// TIA Portal project "VisionSensorKonveyorBandSistemi" (V17)
// Vorlageprojekt für das Buch mit Zielsystem S7-1200

(* hardware
DEVICE "S7-1200-Station_1"  S7-1200 Station
   slot 0: "Baugruppenträger_0"  Rack  V1.0
   slot 1: "PLC_1"  CPU 1211C DC/DC/DC  6ES7 211-1AE40-0XB0  V4.1
*)

// ===== PLC "PLC_1"  CPU 1211C DC/DC/DC =====

VAR_GLOBAL   // PLC tag table "Standard-Variablentabelle"
   "ENTRY CONVEYOR" AT %A0.0 : Bool;
   "EXİT" AT %E0.0 : Bool;
   "START PB" AT %E0.1 : Bool;
   "AUTO MANUAL" AT %I0.5 : Bool;
   "MANUAL" AT %M0.1 : Bool;
   "AUTO" AT %M0.0 : Bool;
   "ONS" AT %M1.1 : Bool;
   "START ONS" AT %M0.3 : Bool;
   "STOP PB" AT %I0.3 : Bool;
   "Tag_3" AT %I0.4 : Bool;
   "RUN MODE" AT %M0.4 : Bool;
   "START LIGHT" AT %Q1.1 : Bool;
   "STOP LIGHT" AT %Q1.3 : Bool;
   "RESET PB" AT %I0.2 : Bool;
   "RESET" AT %M0.2 : Bool;
   "RESET LIGHT" AT %Q1.2 : Bool;
   "VİSİON SENSOR" AT %IW104 : Int;
   "VİSİON SENSOR ARALIK" AT %M1.0 : Bool;
   "STOP ENTRY CONVEYOR" AT %M1.2 : Bool;
   "PRODUCT BLUE OR GREEN" AT %M0.5 : Bool;
   "BLUE BASE OR LID" AT %M0.6 : Bool;
   "GREEN BASE OR LİD" AT %M0.7 : Bool;
   "SORTER 2 BELT" AT %Q0.6 : Bool;
   "SORTER 2TURN" AT %Q0.5 : Bool;
   "Tag_2" AT %QW32 : Int;
   "EXİT CONVEYOR" AT %Q0.2 : Bool;
   "SORTER 1 BELT" AT %Q0.4 : Bool;
   "SORTER 1 TURN" AT %Q0.3 : Bool;
   "Tag_1" AT %QW30 : Int;
   "SORTER 3 BELT" AT %Q1.0 : Bool;
   "SORTER 3 TURN" AT %Q0.7 : Bool;
   "Tag_4" AT %QW34 : Int;
   "VISION SENSOR" AT %IW30 : Word;
END_VAR

// folder: System blocks/Program resources

DATA_BLOCK "IEC_Timer_0_DB"   // DB1
{ S7_Optimized_Access := 'TRUE' }
AUTHOR : Simatic
FAMILY : IEC
NAME : IEC_TMR
VERSION : 1.0
// stored: InstanceOfName IEC_TIMER
"IEC_TIMER"
BEGIN
END_DATA_BLOCK

DATA_BLOCK "IEC_Timer_0_DB_1"   // DB2
{ S7_Optimized_Access := 'TRUE' }
AUTHOR : Simatic
FAMILY : IEC
NAME : IEC_TMR
VERSION : 1.0
// stored: InstanceOfName IEC_TIMER
"IEC_TIMER"
BEGIN
END_DATA_BLOCK

DATA_BLOCK "IEC_Counter_0_DB"   // DB3
{ S7_Optimized_Access := 'TRUE' }
AUTHOR : Simatic
FAMILY : IEC
NAME : CNTR
VERSION : 1.0
// stored: InstanceOfName IEC_COUNTER
"IEC_COUNTER"
BEGIN
END_DATA_BLOCK

DATA_BLOCK "IEC_Counter_0_DB_1"   // DB4
{ S7_Optimized_Access := 'TRUE' }
AUTHOR : Simatic
FAMILY : IEC
NAME : CNTR
VERSION : 1.0
// stored: InstanceOfName IEC_COUNTER
"IEC_COUNTER"
BEGIN
END_DATA_BLOCK

DATA_BLOCK "IEC_Counter_0_DB_2"   // DB5
{ S7_Optimized_Access := 'TRUE' }
AUTHOR : Simatic
FAMILY : IEC
NAME : CNTR
VERSION : 1.0
// stored: InstanceOfName IEC_COUNTER
"IEC_COUNTER"
BEGIN
END_DATA_BLOCK

// folder: (top level)

FUNCTION "MHJ-PLC-Lab-Function-S71200" : Void   // FC9000, SCL
{ S7_Optimized_Access := 'TRUE' }
VERSION : 0.1
   VAR_TEMP
      rdTimeReturn : Int;
      outputTime : DTL;
      SyncVal : Byte;
      forVal : Int;
      forVal_2 : Int;
      Value : Byte;
   END_VAR
   VAR CONSTANT
      CompVal : Byte := 16#34;
      Value_01 : Byte := 16#11;
      Value_01_DW : DWord := 16#A165_D992;
      Value_02_DW : DWord := 16#58BE_4401;
   END_VAR
BEGIN

   #Value:=PEEK(area := 16#82,
        dbNumber := 0,
        byteOffset := 511);
   #Value := #Value + 1;

   POKE(area := 16#82,
        dbNumber := 0,
        byteOffset := 511,
        value := #Value);

   POKE(area:=16#81,
        dbNumber:=0,
        byteOffset:=1016,
        value:=#Value_01_DW);
   POKE(area := 16#81,
        dbNumber := 0,
        byteOffset := 1020,
        value := #Value_02_DW);

   POKE(area := 16#81,
        dbNumber := 0,
        byteOffset := 511,
        value := B#16#00);

   FOR #forVal := 0 TO 120 DO
       FOR #forVal_2:=0 TO 10 DO
           #rdTimeReturn:=RD_SYS_T(#outputTime);
           #rdTimeReturn := WR_SYS_T(#outputTime);
           #rdTimeReturn := RD_SYS_T(#outputTime);
           #rdTimeReturn := WR_SYS_T(#outputTime);
       END_FOR;
       #SyncVal:= PEEK(area := 16#81,
                      dbNumber := 0,
                      byteOffset := 511);
       IF #SyncVal = #CompVal THEN
          GOTO M_1;
       END_IF;
   END_FOR;
   RETURN;

   M_1:
   POKE(area := 16#81,
        dbNumber := 0,
        byteOffset := 511,
        value := B#16#0);
END_FUNCTION

ORGANIZATION_BLOCK "Main"   // OB1, LAD, ProgramCycle
TITLE = "Main Program Sweep (Cycle)"
{ S7_Optimized_Access := 'TRUE' }
VERSION : 0.1
   VAR_INPUT
      Initial_Call : Bool;   // Initial call of this OB
      Remanence : Bool;   // =True, if remanent data are available
   END_VAR
   VAR_TEMP   // added for the SCL form of the ladder/FBD networks
      _w1 : Bool;
      _w2 : Bool;
   END_VAR
BEGIN

REGION Network 1: Konnektierungsbaustein für PLC-Lab
   // Im Netzwerk 1 wird der Konnektierungsbaustein für PLC-Lab aufgerufen.
   // Dieser Aufruf darf nicht entfernt werden!
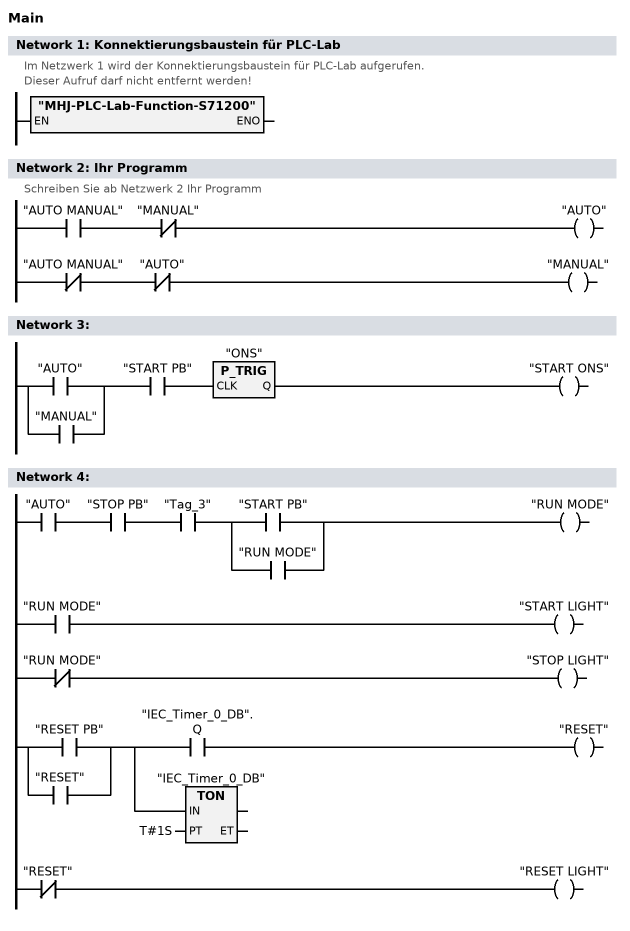
   RUNG wire#powerrail
      "MHJ-PLC-Lab-Function-S71200"()
   END_RUNG
   // the same network as SCL:
   "MHJ-PLC-Lab-Function-S71200"();
END_REGION

REGION Network 2: Ihr Programm
   // Schreiben Sie ab Netzwerk 2 Ihr Programm
   RUNG wire#powerrail
      Contact( "AUTO MANUAL" )
      I_Contact( "MANUAL" )
      Coil( "AUTO" )
   END_RUNG
   RUNG wire#powerrail
      I_Contact( "AUTO MANUAL" )
      I_Contact( "AUTO" )
      Coil( "MANUAL" )
   END_RUNG
   // the same network as SCL:
   "AUTO" := "AUTO MANUAL" AND NOT "MANUAL";
   "MANUAL" := NOT "AUTO MANUAL" AND NOT "AUTO";
END_REGION

REGION Network 3
   RUNG wire#powerrail
      Contact( "AUTO" )
      wire#w1
      Contact( "START PB" )
      P_Trig( "ONS" )
      Coil( "START ONS" )
   END_RUNG
   RUNG wire#powerrail
      Contact( "MANUAL" )
   END_RUNG wire#w1
   // the same network as SCL:
   #_w1 := ("AUTO" OR "MANUAL") AND "START PB";
   #_w2 := #_w1 AND NOT "ONS";   // rising edge
   "ONS" := #_w1;
   "START ONS" := #_w2;
END_REGION

REGION Network 4
   "RUN MODE" := "AUTO" AND "STOP PB" AND "Tag_3" AND ("START PB" OR "RUN MODE");
   "START LIGHT" := "RUN MODE";
   "STOP LIGHT" := NOT "RUN MODE";
   #_w1 := "RESET PB" OR "RESET";
   "RESET" := #_w1 AND "IEC_Timer_0_DB".Q;
   "IEC_Timer_0_DB".TON(IN := #_w1, PT := T#1S);
   "RESET LIGHT" := NOT "RESET";
END_REGION
END_ORGANIZATION_BLOCK

ORGANIZATION_BLOCK "INPUTS"   // OB123, LAD, ProgramCycle
TITLE = "Main Program Sweep (Cycle)"
{ S7_Optimized_Access := 'TRUE' }
VERSION : 0.1
   VAR_INPUT
      Initial_Call : Bool;   // Initial call of this OB
      Remanence : Bool;   // =True, if remanent data are available
   END_VAR
BEGIN

REGION Network 1
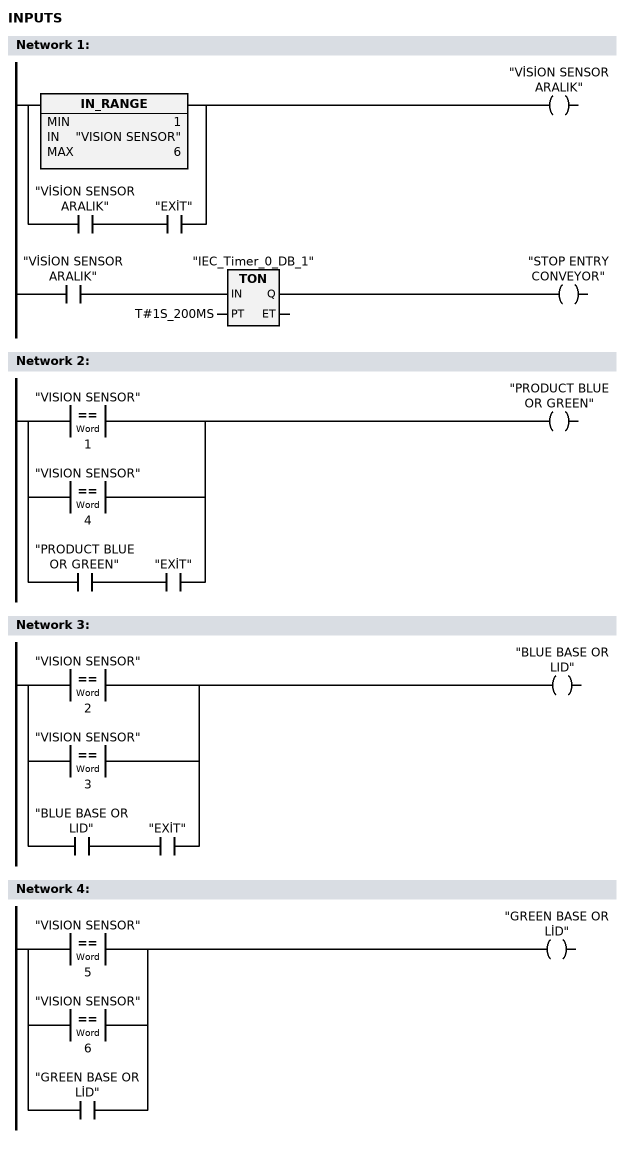
   "VİSİON SENSOR ARALIK" := ((1 <= "VISION SENSOR") AND ("VISION SENSOR" <= 6)) OR ("VİSİON SENSOR ARALIK" AND "EXİT");
   "IEC_Timer_0_DB_1".TON(IN := "VİSİON SENSOR ARALIK", PT := T#1S_200MS);
   "STOP ENTRY CONVEYOR" := "IEC_Timer_0_DB_1".Q;
END_REGION

REGION Network 2
   RUNG wire#powerrail
      { S7_Templates := "SrcType := Word" } EQ_Contact(in1 := "VISION SENSOR", in2 := 1)
      wire#w1
      Coil( "PRODUCT BLUE OR GREEN" )
   END_RUNG
   RUNG wire#powerrail
      { S7_Templates := "SrcType := Word" } EQ_Contact(in1 := "VISION SENSOR", in2 := 4)
   END_RUNG wire#w1
   RUNG wire#powerrail
      Contact( "PRODUCT BLUE OR GREEN" )
      Contact( "EXİT" )
   END_RUNG wire#w1
   // the same network as SCL:
   "PRODUCT BLUE OR GREEN" := ("VISION SENSOR" = 1) OR ("VISION SENSOR" = 4) OR ("PRODUCT BLUE OR GREEN" AND "EXİT");
END_REGION

REGION Network 3
   RUNG wire#powerrail
      { S7_Templates := "SrcType := Word" } EQ_Contact(in1 := "VISION SENSOR", in2 := 2)
      wire#w1
      Coil( "BLUE BASE OR LID" )
   END_RUNG
   RUNG wire#powerrail
      { S7_Templates := "SrcType := Word" } EQ_Contact(in1 := "VISION SENSOR", in2 := 3)
   END_RUNG wire#w1
   RUNG wire#powerrail
      Contact( "BLUE BASE OR LID" )
      Contact( "EXİT" )
   END_RUNG wire#w1
   // the same network as SCL:
   "BLUE BASE OR LID" := ("VISION SENSOR" = 2) OR ("VISION SENSOR" = 3) OR ("BLUE BASE OR LID" AND "EXİT");
END_REGION

REGION Network 4
   RUNG wire#powerrail
      { S7_Templates := "SrcType := Word" } EQ_Contact(in1 := "VISION SENSOR", in2 := 5)
      wire#w1
      Coil( "GREEN BASE OR LİD" )
   END_RUNG
   RUNG wire#powerrail
      { S7_Templates := "SrcType := Word" } EQ_Contact(in1 := "VISION SENSOR", in2 := 6)
   END_RUNG wire#w1
   RUNG wire#powerrail
      Contact( "GREEN BASE OR LİD" )
   END_RUNG wire#w1
   // the same network as SCL:
   "GREEN BASE OR LİD" := ("VISION SENSOR" = 5) OR ("VISION SENSOR" = 6) OR "GREEN BASE OR LİD";
END_REGION
END_ORGANIZATION_BLOCK

ORGANIZATION_BLOCK "OUTPUTS"   // OB124, LAD, ProgramCycle
TITLE = "Main Program Sweep (Cycle)"
{ S7_Optimized_Access := 'TRUE' }
VERSION : 0.1
   VAR_INPUT
      Initial_Call : Bool;   // Initial call of this OB
      Remanence : Bool;   // =True, if remanent data are available
   END_VAR
BEGIN

REGION Network 1
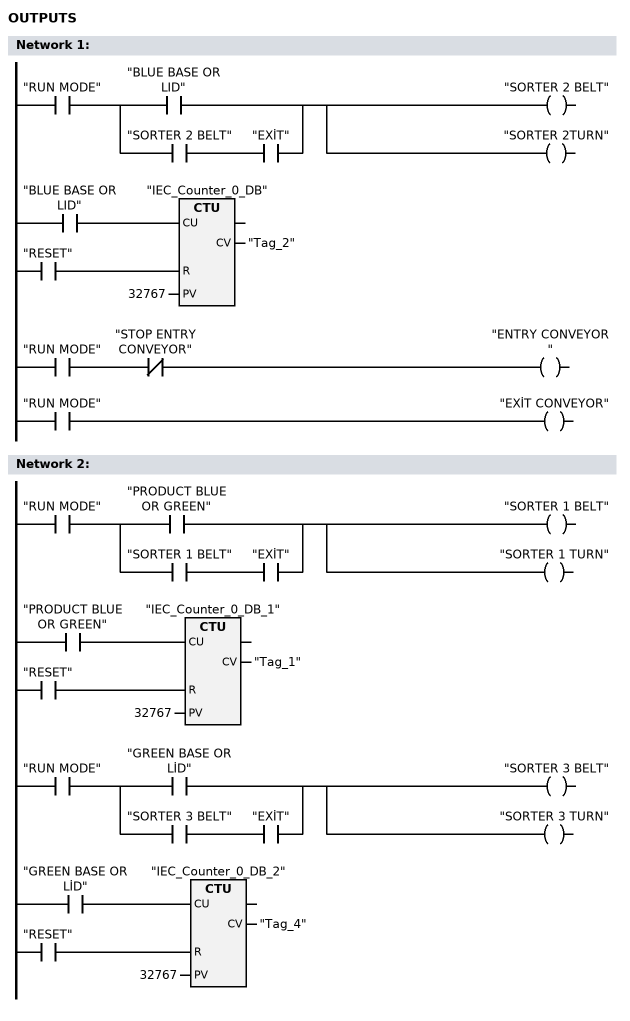
   "SORTER 2 BELT" := "RUN MODE" AND ("BLUE BASE OR LID" OR ("SORTER 2 BELT" AND "EXİT"));
   "SORTER 2TURN" := "SORTER 2 BELT";
   "IEC_Counter_0_DB".CTU(CU := "BLUE BASE OR LID", R := "RESET", PV := 32767, CV => "Tag_2");
   "ENTRY CONVEYOR" := "RUN MODE" AND NOT "STOP ENTRY CONVEYOR";
   "EXİT CONVEYOR" := "RUN MODE";
END_REGION

REGION Network 2
   "SORTER 1 BELT" := "RUN MODE" AND ("PRODUCT BLUE OR GREEN" OR ("SORTER 1 BELT" AND "EXİT"));
   "SORTER 1 TURN" := "SORTER 1 BELT";
   "IEC_Counter_0_DB_1".CTU(CU := "PRODUCT BLUE OR GREEN", R := "RESET", PV := 32767, CV => "Tag_1");
   "SORTER 3 BELT" := "RUN MODE" AND ("GREEN BASE OR LİD" OR ("SORTER 3 BELT" AND "EXİT"));
   "SORTER 3 TURN" := "SORTER 3 BELT";
   "IEC_Counter_0_DB_2".CTU(CU := "GREEN BASE OR LİD", R := "RESET", PV := 32767, CV => "Tag_4");
END_REGION
END_ORGANIZATION_BLOCK